// TIA Portal V19 export
DATA_BLOCK "RECIPE DB"   // DB9
{ S7_Optimized_Access := 'FALSE' }
   VAR
      "RINSE-1_CLEANING_TIME_SV" : Int;
      "RINSE-1_RECIRCULATION_TIME_SV" : Int;
      "RINSE-1_DRAIN_TIME_SV" : Int;
      "RINSE-1_PUMP_CHASING_TIME_SV" : Int;
      "RINSE-1_TEMPERATURE_SET" : Real;
      "RINSE-1_FWD_PUMP_HEATING_RPM" : Int;
      "RINSE-1_FWD_PUMP_CLEANING_RPM" : Int;
      "RINSE-2_TEMPERATURE_SET" : Real;
      "RINSE-2_CLEANING_TIME_SV" : Int;
      "RINSE-2_RECIRCULATION_TIME_SV" : Int;
      "RINSE-2_DRAIN_TIME_SV" : Int;
      "RINSE-2_PUMP_CHASING_TIME_SV" : Int;
      "RINSE-2_FWD_PUMP_HEATING_RPM" : Int;
      "RINSE-2_FWD_PUMP_CLEANING_RPM" : Int;
      DOSING_TIME_SV : Int;
      "ALKALI/ACID_TEMPERATURE_SET" : Real;
      "ALKALI/ACID_CLEANING_TIME_SV" : Int;
      "ALKALI/ACID_RECIRCULATION_TIME_SV" : Int;
      "ALKALI/ACID_DRAIN_TIME_SV" : Int;
      "ALKALI/ACID_PUMP_CHASING_TIME_SV" : Int;
      "ALKALI/ACID_FWD_PUMP_HEATING_RPM" : Int;
      "ALKALI/ACID_FWD_PUMP_CLEANING_RPM" : Int;
      FINAL_RINSE_TEMPERATURE_SET : Real;
      FINAL_RINSE_CLEANING_TIME_SV : Int;
      FINAL_RINSE_RECIRCULATION_TIME_SV : Int;
      FINAL_RINSE_DRAIN_TIME_SV : Int;
      FINAL_RINSE_PUMP_CHASING_TIME_SV : Int;
      "FINAL_RINSE-2_FWD_PUMP_HEATING_RPM" : Int;
      "FINAL_RINSE-2_FWD_PUMP_CLEANING_RPM" : Int;
      CONDUCTIVITY_SET : Real;
      "PH_SET (NOT USED)" : Int;
      DOSING_PH_LOW : Real;
      DOSING_PH_HIGH : Real;
      "RINSE-3_TEMPERATURE_SET" : Real;
      "RINSE-3_CLEANING_TIME_SV" : Int;
      "RINSE-3_RECIRCULATION_TIME_SV" : Int;
      "RINSE-3_DRAIN_TIME_SV" : Int;
      "RINSE-3_PUMP_CHASING_TIME_SV" : Int;
      "FINAL_RINSE-1_FWD_PUMP_HEATING_RPM" : Int;
      "FINAL_RINSE-1_FWD_PUMP_CLEANING_RPM" : Int;
      SET_TEMPERATURE : Real;
      "RINSE-1_SELECT" : Bool;
      "ALKALI / ACID_SELECT" : Bool;
      "RINSE-2_SELECT" : Bool;
      "FINAL_RINSE-1_SELECT" : Bool;
      "FINAL_RINSE-2_SELECT" : Bool;
      RECIRCULATION_PH_LOW : Real;
      RECIRCULATION_PH_HIGH : Real;
      "SW TANK_SELECT" : Bool;
      "PW TANK_SELECT" : Bool;
      "SW TANK_FWD_PUMP_CLEANING_RPM" : Int;
      "PW TANK_FWD_PUMP_CLEANING_RPM" : Int;
      "SW TANK_TEMPERATURE_SET" : Real;
      "PW TANK_TEMPERATURE_SET" : Real;
      "SW TANK_CLEANING_TIME_SV" : Int;
      "SW TANK_DRAIN_TIME_SV" : Int;
      "SW TANK_PUMP_CHASING_TIME_SV" : Int;
      "PW TANK_CLEANING_TIME_SV" : Int;
      "PW TANK_DRAIN_TIME_SV" : Int;
      "PW TANK_PUMP_CHASING_TIME_SV" : Int;
   END_VAR
BEGIN
END_DATA_BLOCK
